(* PLC project poST.project, poSTIDE *)
(* stored: creationDateTime 2021-08-31T00:00:00.000000 *)

FUNCTION SUB : ANY_MAGNITUDE
  VAR_INPUT
    in1 : ANY_MAGNITUDE;
    in2 : ANY_MAGNITUDE;
  END_VAR

END_FUNCTION
